# EPICS substitutions: backup/mc12/tpmacApp/Db/pmac_asyn_motor.substitutions
file "db/pmac_asyn_motor.db"
{

pattern
{SYS,              DEV,                 MOTOR,  SPORT,  ADDR,  DESC,        DTYP        PREC,  EGU }
{"XF:23ID1-OP",    "{Dif-Ax:Del}",      "motor", "P0",    1,    "Delta",    "asynMotor",  4,      "deg" }
{"XF:23ID1-OP",    "{Dif-Ax:Th}",      "motor", "P0",    2,    "Theta",     "asynMotor",  4,      "deg" }
{"XF:23ID1-OP",    "{Dif-Ax:Gam}",      "motor", "P0",    3,    "Gamma",    "asynMotor",  4,      "deg" }
{"XF:23ID1-OP",    "{Dif-Ax:MuR}",      "motor", "P0",    4,    "Mu Rotation","asynMotor",  4,    "deg" }
{"XF:23ID1-OP",    "{Dif-Ax:MuT}",      "motor", "P0",    5,    "Mu Translation","asynMotor",  4, "mm" }
{"XF:23ID1-OP",    "{Dif-Ax:XS}",      "motor", "P0",    6,    "Sample X",  "asynMotor",  4,      "mm" }
{"XF:23ID1-OP",    "{Dif-Ax:YS}",      "motor", "P0",    7,    "Sample Y",  "asynMotor",  4,      "mm" }
{"XF:23ID1-OP",    "{Dif-Ax:ZS}",      "motor", "P0",    8,    "Sample Z",  "asynMotor",  4,      "mm" }

}
